PROGRAM PRG_Test
VAR
	fbSaMControllerTest				: FB_SaMControllerTest;
	fbMachineControlTest			: FB_MachineControl_NoneTE_Test;
	
END_VAR


	TcUnit.RUN_IN_SEQUENCE ();

END_PROGRAM

(* stored: Version 1.1.0.1, ProductVersion 3.1.4024.15
   POU PRG_Test: Id {d2be5eed-9005-4536-8d51-b8ea05870e24}, SpecialFunc None *)
